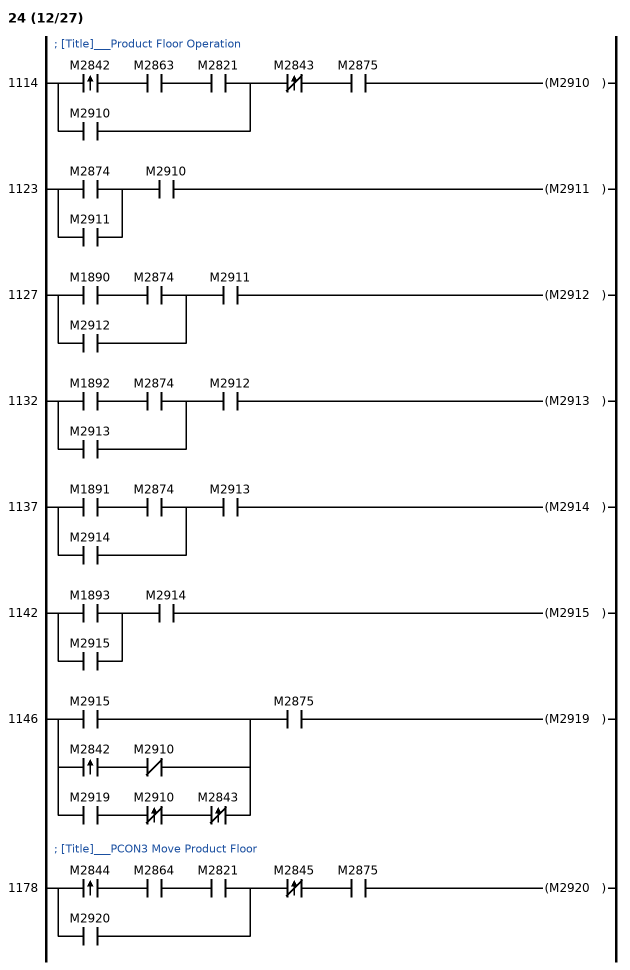
; [Title]___Product Floor Operation
1114  LDP     M2842
      AND     M2863
      AND     M2821
      OR      M2910
      ANDPI   M2843
      AND     M2875
      OUT     M2910
1123  LD      M2874
      OR      M2911
      AND     M2910
      OUT     M2911
1127  LD      M1890
      AND     M2874
      OR      M2912
      AND     M2911
      OUT     M2912
1132  LD      M1892
      AND     M2874
      OR      M2913
      AND     M2912
      OUT     M2913
1137  LD      M1891
      AND     M2874
      OR      M2914
      AND     M2913
      OUT     M2914
1142  LD      M1893
      OR      M2915
      AND     M2914
      OUT     M2915
1146  LD      M2915
      LDP     M2842
      ANI     M2910
      ORB
      LD      M2919
      ANDPI   M2910
      ANDPI   M2843
      ORB
      AND     M2875
      OUT     M2919
; [Title]___PCON3 Move Product Floor
1178  LDP     M2844
      AND     M2864
      AND     M2821
      OR      M2920
      ANDPI   M2845
      AND     M2875
      OUT     M2920
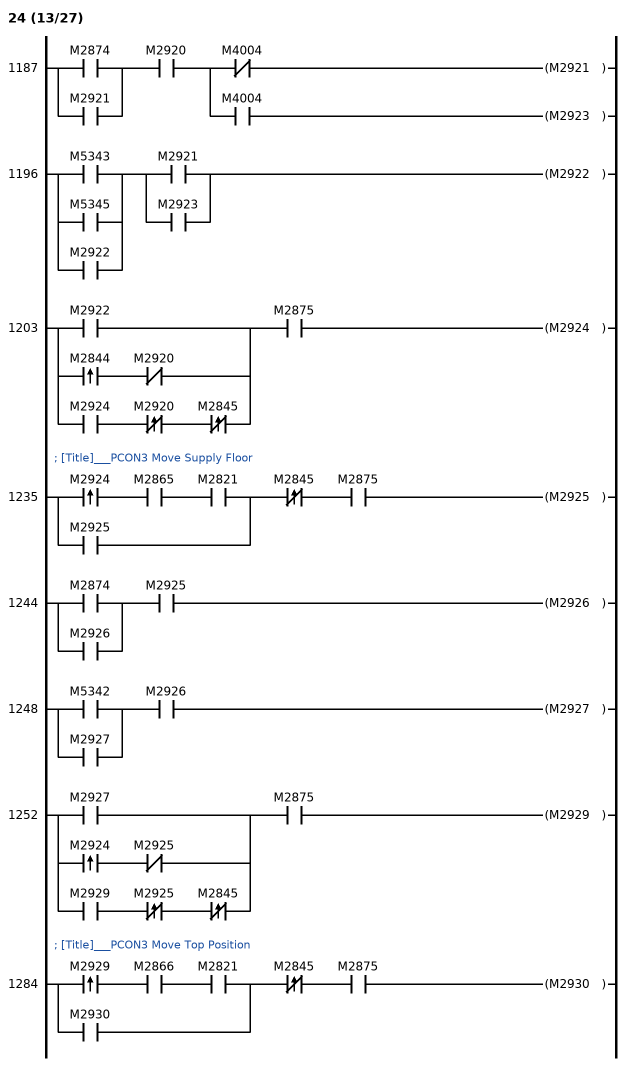
1187  LD      M2874
      OR      M2921
      AND     M2920
      MPS
      ANI     M4004
      OUT     M2921
      MPP
      AND     M4004
      OUT     M2923
1196  LD      M5343
      OR      M5345
      OR      M2922
      LD      M2921
      OR      M2923
      ANB
      OUT     M2922
1203  LD      M2922
      LDP     M2844
      ANI     M2920
      ORB
      LD      M2924
      ANDPI   M2920
      ANDPI   M2845
      ORB
      AND     M2875
      OUT     M2924
; [Title]___PCON3 Move Supply Floor
1235  LDP     M2924
      AND     M2865
      AND     M2821
      OR      M2925
      ANDPI   M2845
      AND     M2875
      OUT     M2925
1244  LD      M2874
      OR      M2926
      AND     M2925
      OUT     M2926
1248  LD      M5342
      OR      M2927
      AND     M2926
      OUT     M2927
1252  LD      M2927
      LDP     M2924
      ANI     M2925
      ORB
      LD      M2929
      ANDPI   M2925
      ANDPI   M2845
      ORB
      AND     M2875
      OUT     M2929
; [Title]___PCON3 Move Top Position
1284  LDP     M2929
      AND     M2866
      AND     M2821
      OR      M2930
      ANDPI   M2845
      AND     M2875
      OUT     M2930
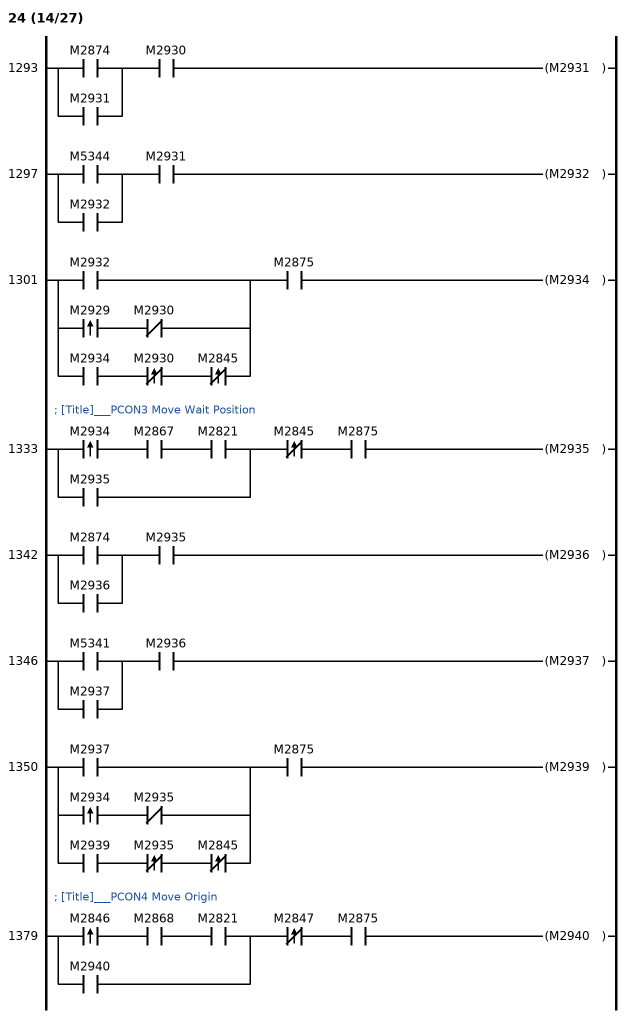
1293  LD      M2874
      OR      M2931
      AND     M2930
      OUT     M2931
1297  LD      M5344
      OR      M2932
      AND     M2931
      OUT     M2932
1301  LD      M2932
      LDP     M2929
      ANI     M2930
      ORB
      LD      M2934
      ANDPI   M2930
      ANDPI   M2845
      ORB
      AND     M2875
      OUT     M2934
; [Title]___PCON3 Move Wait Position
1333  LDP     M2934
      AND     M2867
      AND     M2821
      OR      M2935
      ANDPI   M2845
      AND     M2875
      OUT     M2935
1342  LD      M2874
      OR      M2936
      AND     M2935
      OUT     M2936
1346  LD      M5341
      OR      M2937
      AND     M2936
      OUT     M2937
1350  LD      M2937
      LDP     M2934
      ANI     M2935
      ORB
      LD      M2939
      ANDPI   M2935
      ANDPI   M2845
      ORB
      AND     M2875
      OUT     M2939
; [Title]___PCON4 Move Origin
1379  LDP     M2846
      AND     M2868
      AND     M2821
      OR      M2940
      ANDPI   M2847
      AND     M2875
      OUT     M2940
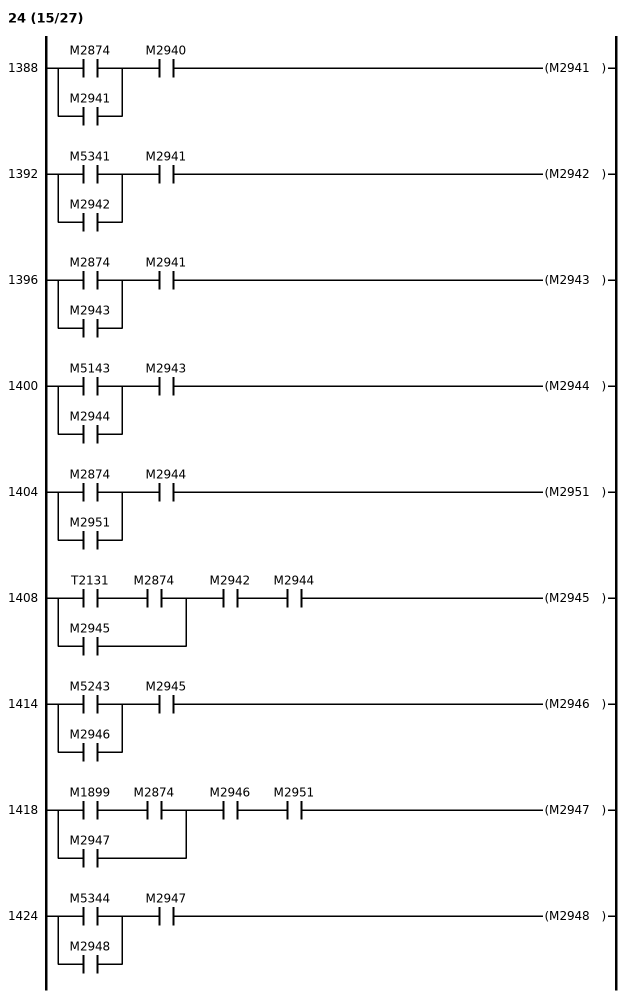
1388  LD      M2874
      OR      M2941
      AND     M2940
      OUT     M2941
1392  LD      M5341
      OR      M2942
      AND     M2941
      OUT     M2942
1396  LD      M2874
      OR      M2943
      AND     M2941
      OUT     M2943
1400  LD      M5143
      OR      M2944
      AND     M2943
      OUT     M2944
1404  LD      M2874
      OR      M2951
      AND     M2944
      OUT     M2951
1408  LD      T2131
      AND     M2874
      OR      M2945
      AND     M2942
      AND     M2944
      OUT     M2945
1414  LD      M5243
      OR      M2946
      AND     M2945
      OUT     M2946
1418  LD      M1899
      AND     M2874
      OR      M2947
      AND     M2946
      AND     M2951
      OUT     M2947
1424  LD      M5344
      OR      M2948
      AND     M2947
      OUT     M2948
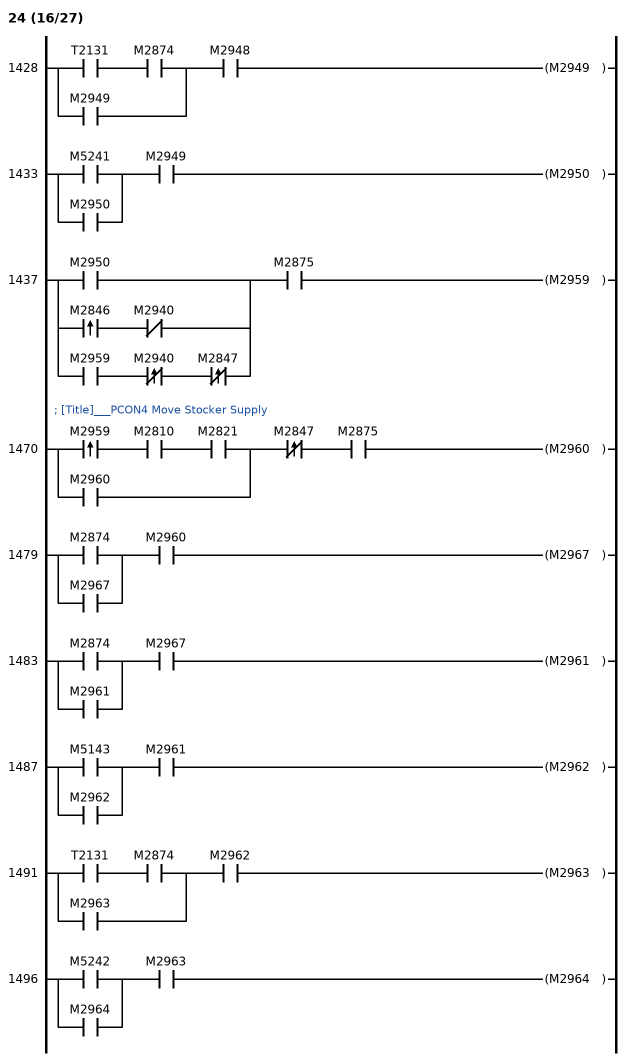
1428  LD      T2131
      AND     M2874
      OR      M2949
      AND     M2948
      OUT     M2949
1433  LD      M5241
      OR      M2950
      AND     M2949
      OUT     M2950
1437  LD      M2950
      LDP     M2846
      ANI     M2940
      ORB
      LD      M2959
      ANDPI   M2940
      ANDPI   M2847
      ORB
      AND     M2875
      OUT     M2959
; [Title]___PCON4 Move Stocker Supply
1470  LDP     M2959
      AND     M2810
      AND     M2821
      OR      M2960
      ANDPI   M2847
      AND     M2875
      OUT     M2960
1479  LD      M2874
      OR      M2967
      AND     M2960
      OUT     M2967
1483  LD      M2874
      OR      M2961
      AND     M2967
      OUT     M2961
1487  LD      M5143
      OR      M2962
      AND     M2961
      OUT     M2962
1491  LD      T2131
      AND     M2874
      OR      M2963
      AND     M2962
      OUT     M2963
1496  LD      M5242
      OR      M2964
      AND     M2963
      OUT     M2964
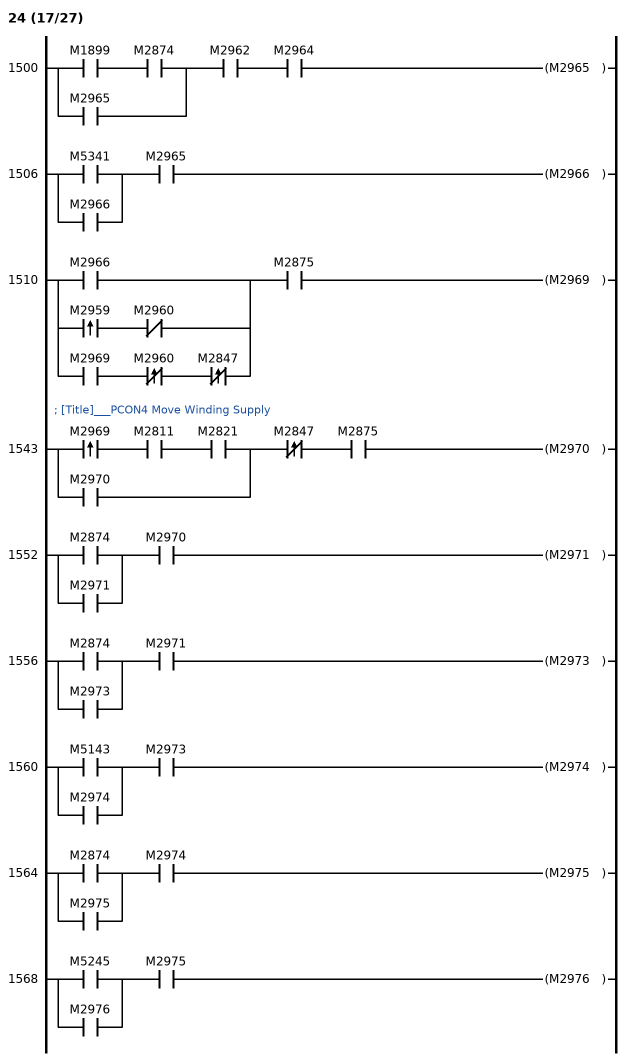
1500  LD      M1899
      AND     M2874
      OR      M2965
      AND     M2962
      AND     M2964
      OUT     M2965
1506  LD      M5341
      OR      M2966
      AND     M2965
      OUT     M2966
1510  LD      M2966
      LDP     M2959
      ANI     M2960
      ORB
      LD      M2969
      ANDPI   M2960
      ANDPI   M2847
      ORB
      AND     M2875
      OUT     M2969
; [Title]___PCON4 Move Winding Supply
1543  LDP     M2969
      AND     M2811
      AND     M2821
      OR      M2970
      ANDPI   M2847
      AND     M2875
      OUT     M2970
1552  LD      M2874
      OR      M2971
      AND     M2970
      OUT     M2971
1556  LD      M2874
      OR      M2973
      AND     M2971
      OUT     M2973
1560  LD      M5143
      OR      M2974
      AND     M2973
      OUT     M2974
1564  LD      M2874
      OR      M2975
      AND     M2974
      OUT     M2975
1568  LD      M5245
      OR      M2976
      AND     M2975
      OUT     M2976
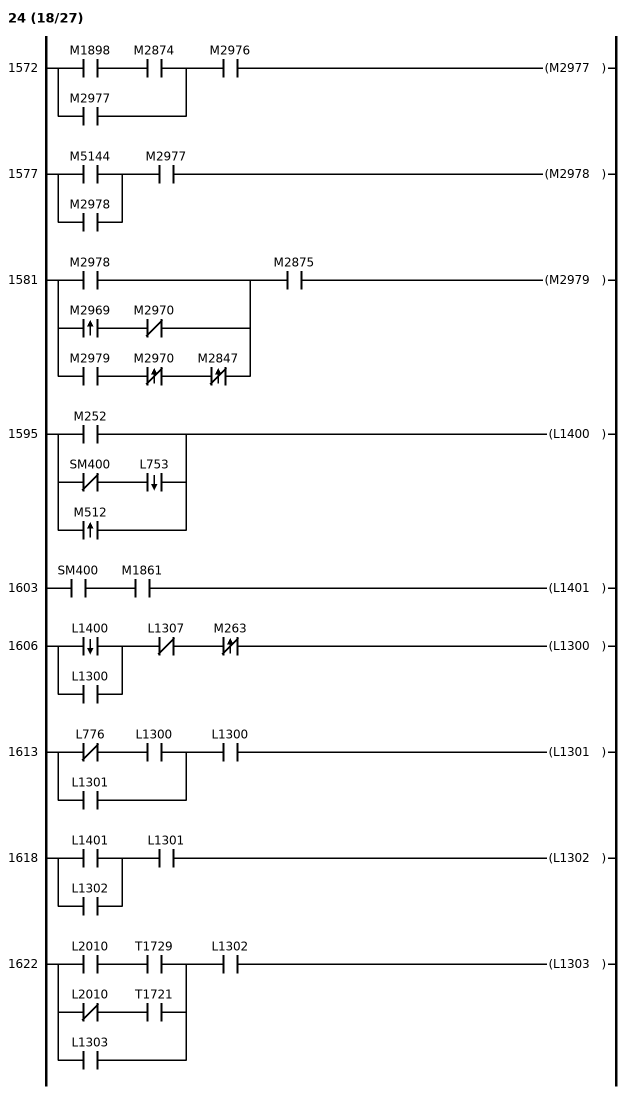
1572  LD      M1898
      AND     M2874
      OR      M2977
      AND     M2976
      OUT     M2977
1577  LD      M5144
      OR      M2978
      AND     M2977
      OUT     M2978
1581  LD      M2978
      LDP     M2969
      ANI     M2970
      ORB
      LD      M2979
      ANDPI   M2970
      ANDPI   M2847
      ORB
      AND     M2875
      OUT     M2979
; 
1595  LD      M252
      LDI     SM400
      ANDF    L753
      ORB
      ORP     M512
      OUT     L1400
1603  LD      SM400
      AND     M1861
      OUT     L1401
1606  LDF     L1400
      OR      L1300
      ANI     L1307
      ANDPI   M263
      OUT     L1300
1613  LDI     L776
      AND     L1300
      OR      L1301
      AND     L1300
      OUT     L1301
1618  LD      L1401
      OR      L1302
      AND     L1301
      OUT     L1302
1622  LD      L2010
      AND     T1729
      LDI     L2010
      AND     T1721
      ORB
      OR      L1303
      AND     L1302
      OUT     L1303
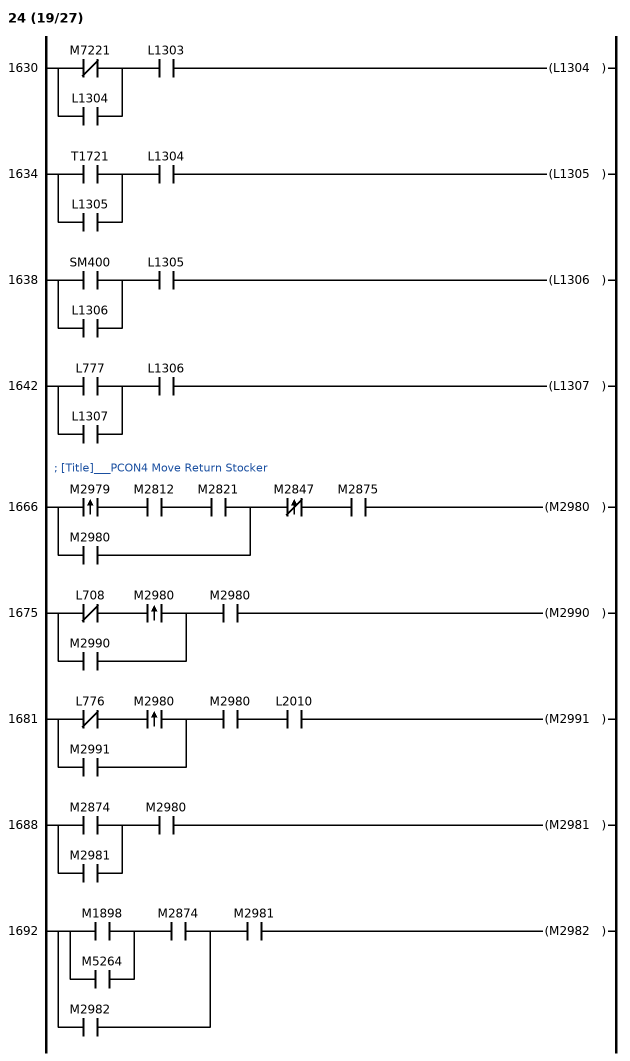
1630  LDI     M7221
      OR      L1304
      AND     L1303
      OUT     L1304
1634  LD      T1721
      OR      L1305
      AND     L1304
      OUT     L1305
1638  LD      SM400
      OR      L1306
      AND     L1305
      OUT     L1306
1642  LD      L777
      OR      L1307
      AND     L1306
      OUT     L1307
; [Title]___PCON4 Move Return Stocker
1666  LDP     M2979
      AND     M2812
      AND     M2821
      OR      M2980
      ANDPI   M2847
      AND     M2875
      OUT     M2980
1675  LDI     L708
      ANDP    M2980
      OR      M2990
      AND     M2980
      OUT     M2990
1681  LDI     L776
      ANDP    M2980
      OR      M2991
      AND     M2980
      AND     L2010
      OUT     M2991
1688  LD      M2874
      OR      M2981
      AND     M2980
      OUT     M2981
1692  LD      M1898
      OR      M5264
      AND     M2874
      OR      M2982
      AND     M2981
      OUT     M2982
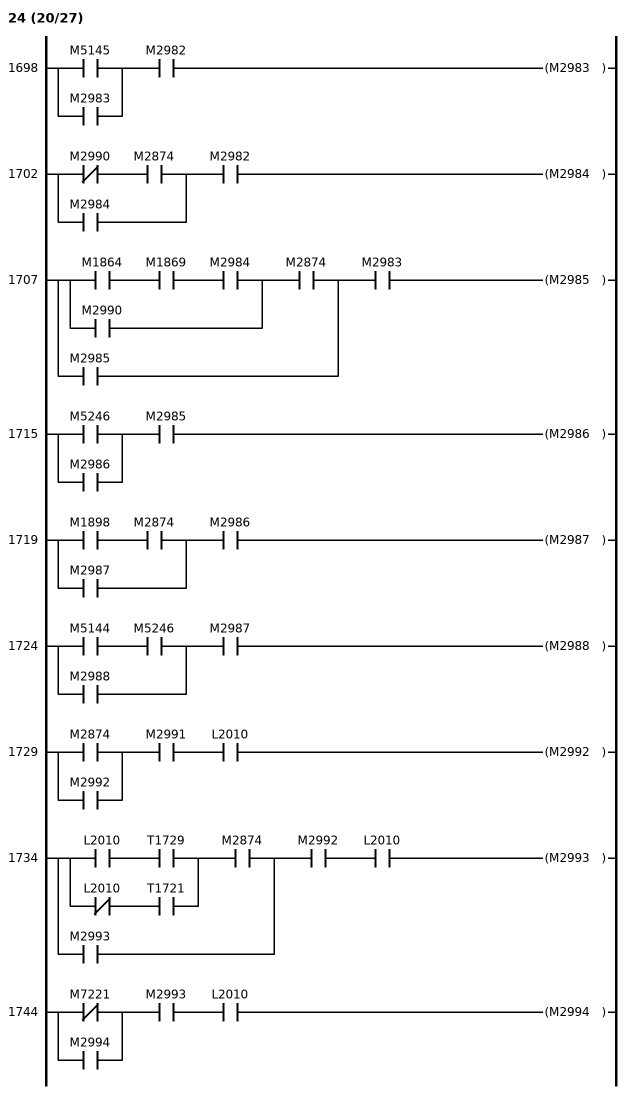
1698  LD      M5145
      OR      M2983
      AND     M2982
      OUT     M2983
1702  LDI     M2990
      AND     M2874
      OR      M2984
      AND     M2982
      OUT     M2984
1707  LD      M1864
      AND     M1869
      AND     M2984
      OR      M2990
      AND     M2874
      OR      M2985
      AND     M2983
      OUT     M2985
1715  LD      M5246
      OR      M2986
      AND     M2985
      OUT     M2986
1719  LD      M1898
      AND     M2874
      OR      M2987
      AND     M2986
      OUT     M2987
1724  LD      M5144
      AND     M5246
      OR      M2988
      AND     M2987
      OUT     M2988
1729  LD      M2874
      OR      M2992
      AND     M2991
      AND     L2010
      OUT     M2992
1734  LD      L2010
      AND     T1729
      LDI     L2010
      AND     T1721
      ORB
      AND     M2874
      OR      M2993
      AND     M2992
      AND     L2010
      OUT     M2993
1744  LDI     M7221
      OR      M2994
      AND     M2993
      AND     L2010
      OUT     M2994
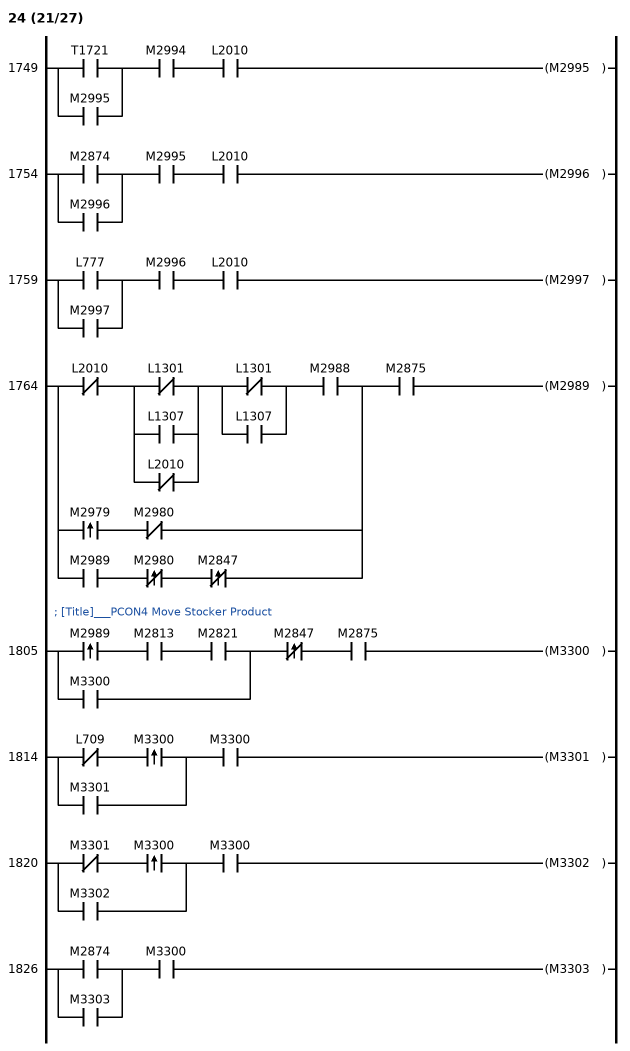
1749  LD      T1721
      OR      M2995
      AND     M2994
      AND     L2010
      OUT     M2995
1754  LD      M2874
      OR      M2996
      AND     M2995
      AND     L2010
      OUT     M2996
1759  LD      L777
      OR      M2997
      AND     M2996
      AND     L2010
      OUT     M2997
1764  LDI     L2010
      LDI     L1301
      OR      L1307
      ORI     L2010
      ANB
      LDI     L1301
      OR      L1307
      ANB
      AND     M2988
      LDP     M2979
      ANI     M2980
      ORB
      LD      M2989
      ANDPI   M2980
      ANDPI   M2847
      ORB
      AND     M2875
      OUT     M2989
; [Title]___PCON4 Move Stocker Product
1805  LDP     M2989
      AND     M2813
      AND     M2821
      OR      M3300
      ANDPI   M2847
      AND     M2875
      OUT     M3300
1814  LDI     L709
      ANDP    M3300
      OR      M3301
      AND     M3300
      OUT     M3301
1820  LDI     M3301
      ANDP    M3300
      OR      M3302
      AND     M3300
      OUT     M3302
1826  LD      M2874
      OR      M3303
      AND     M3300
      OUT     M3303
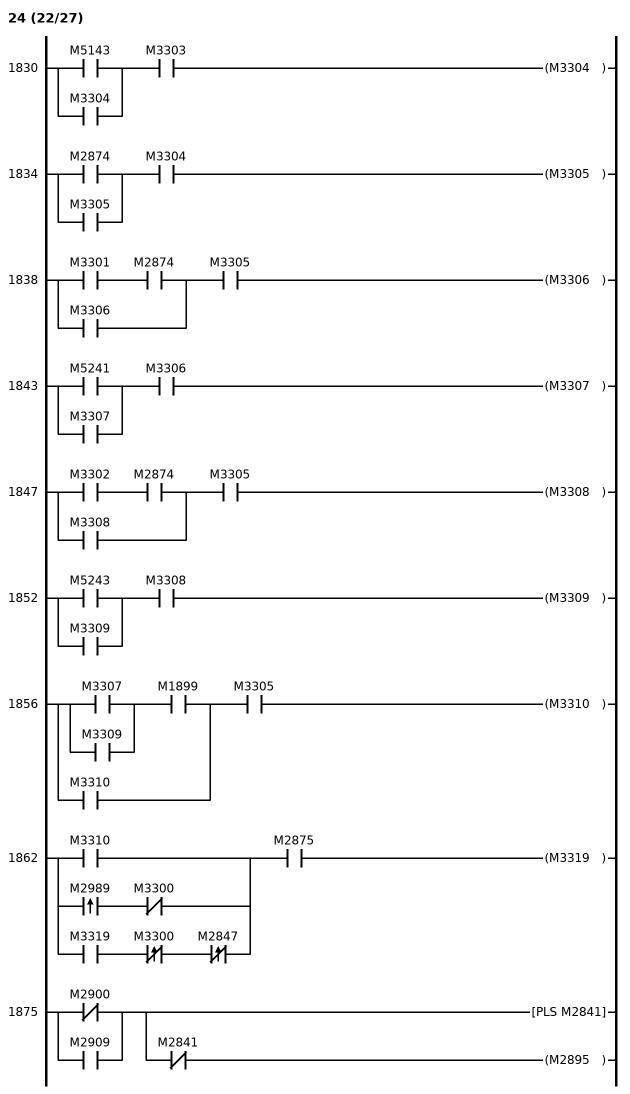
1830  LD      M5143
      OR      M3304
      AND     M3303
      OUT     M3304
1834  LD      M2874
      OR      M3305
      AND     M3304
      OUT     M3305
1838  LD      M3301
      AND     M2874
      OR      M3306
      AND     M3305
      OUT     M3306
1843  LD      M5241
      OR      M3307
      AND     M3306
      OUT     M3307
1847  LD      M3302
      AND     M2874
      OR      M3308
      AND     M3305
      OUT     M3308
1852  LD      M5243
      OR      M3309
      AND     M3308
      OUT     M3309
1856  LD      M3307
      OR      M3309
      AND     M1899
      OR      M3310
      AND     M3305
      OUT     M3310
1862  LD      M3310
      LDP     M2989
      ANI     M3300
      ORB
      LD      M3319
      ANDPI   M3300
      ANDPI   M2847
      ORB
      AND     M2875
      OUT     M3319
1875  LDI     M2900
      OR      M2909
      PLS     M2841
      ANI     M2841
      OUT     M2895
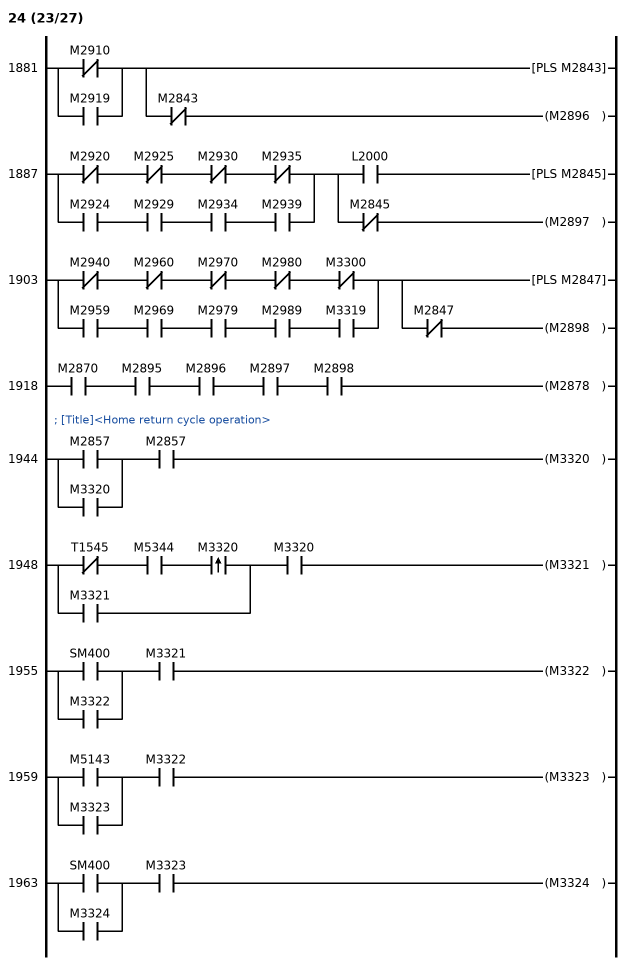
1881  LDI     M2910
      OR      M2919
      PLS     M2843
      ANI     M2843
      OUT     M2896
1887  LDI     M2920
      ANI     M2925
      ANI     M2930
      ANI     M2935
      LD      M2924
      AND     M2929
      AND     M2934
      AND     M2939
      ORB
      MPS
      AND     L2000
      PLS     M2845
      MPP
      ANI     M2845
      OUT     M2897
1903  LDI     M2940
      ANI     M2960
      ANI     M2970
      ANI     M2980
      ANI     M3300
      LD      M2959
      AND     M2969
      AND     M2979
      AND     M2989
      AND     M3319
      ORB
      PLS     M2847
      ANI     M2847
      OUT     M2898
1918  LD      M2870
      AND     M2895
      AND     M2896
      AND     M2897
      AND     M2898
      OUT     M2878
; [Title]<Home return cycle operation>
1944  LD      M2857
      OR      M3320
      AND     M2857
      OUT     M3320
1948  LDI     T1545
      AND     M5344
      ANDP    M3320
      OR      M3321
      AND     M3320
      OUT     M3321
1955  LD      SM400
      OR      M3322
      AND     M3321
      OUT     M3322
1959  LD      M5143
      OR      M3323
      AND     M3322
      OUT     M3323
1963  LD      SM400
      OR      M3324
      AND     M3323
      OUT     M3324
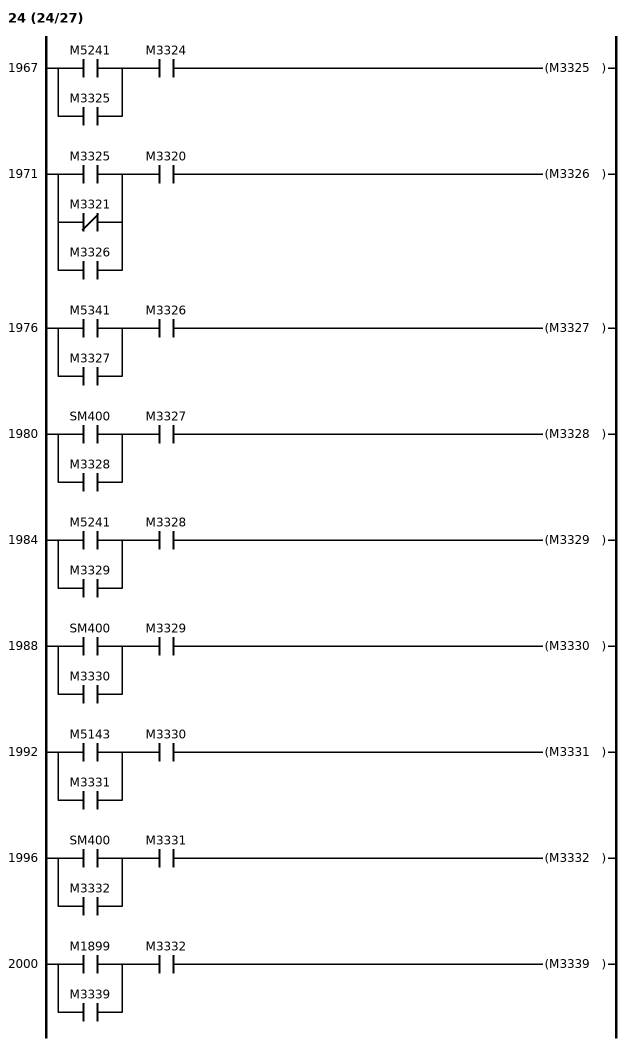
1967  LD      M5241
      OR      M3325
      AND     M3324
      OUT     M3325
1971  LD      M3325
      ORI     M3321
      OR      M3326
      AND     M3320
      OUT     M3326
1976  LD      M5341
      OR      M3327
      AND     M3326
      OUT     M3327
1980  LD      SM400
      OR      M3328
      AND     M3327
      OUT     M3328
1984  LD      M5241
      OR      M3329
      AND     M3328
      OUT     M3329
1988  LD      SM400
      OR      M3330
      AND     M3329
      OUT     M3330
1992  LD      M5143
      OR      M3331
      AND     M3330
      OUT     M3331
1996  LD      SM400
      OR      M3332
      AND     M3331
      OUT     M3332
2000  LD      M1899
      OR      M3339
      AND     M3332
      OUT     M3339
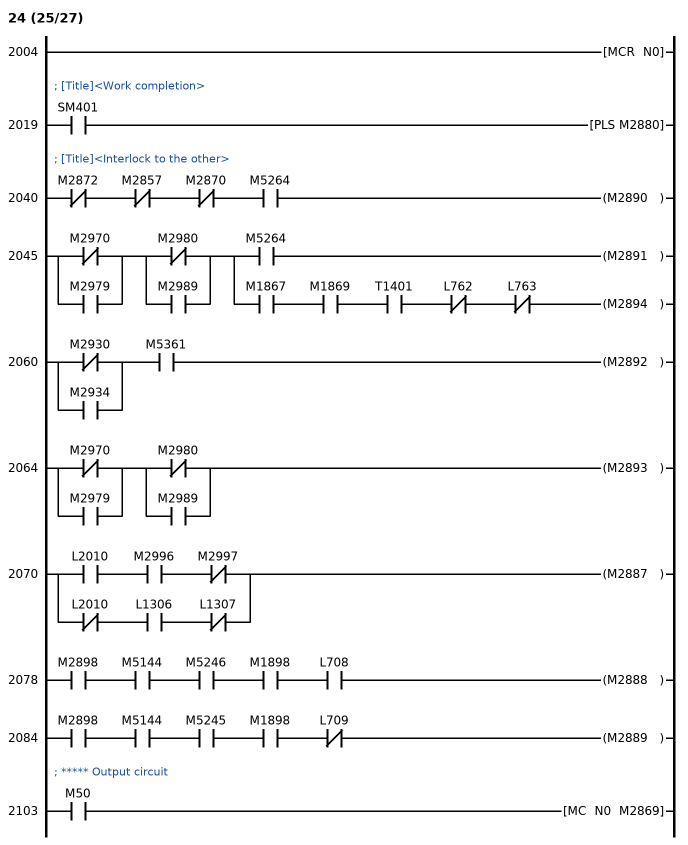
2004  MCR     N0
; [Title]<Work completion>
2019  LD      SM401
      PLS     M2880
; [Title]<Interlock to the other>
2040  LDI     M2872
      ANI     M2857
      ANI     M2870
      AND     M5264
      OUT     M2890
2045  LDI     M2970
      OR      M2979
      LDI     M2980
      OR      M2989
      ANB
      MPS
      AND     M5264
      OUT     M2891
      MPP
      AND     M1867
      AND     M1869
      AND     T1401
      ANI     L762
      ANI     L763
      OUT     M2894
2060  LDI     M2930
      OR      M2934
      AND     M5361
      OUT     M2892
2064  LDI     M2970
      OR      M2979
      LDI     M2980
      OR      M2989
      ANB
      OUT     M2893
2070  LD      L2010
      AND     M2996
      ANI     M2997
      LDI     L2010
      AND     L1306
      ANI     L1307
      ORB
      OUT     M2887
2078  LD      M2898
      AND     M5144
      AND     M5246
      AND     M1898
      AND     L708
      OUT     M2888
2084  LD      M2898
      AND     M5144
      AND     M5245
      AND     M1898
      ANI     L709
      OUT     M2889
; ***** Output circuit
2103  LD      M50
      MC      N0 M2869
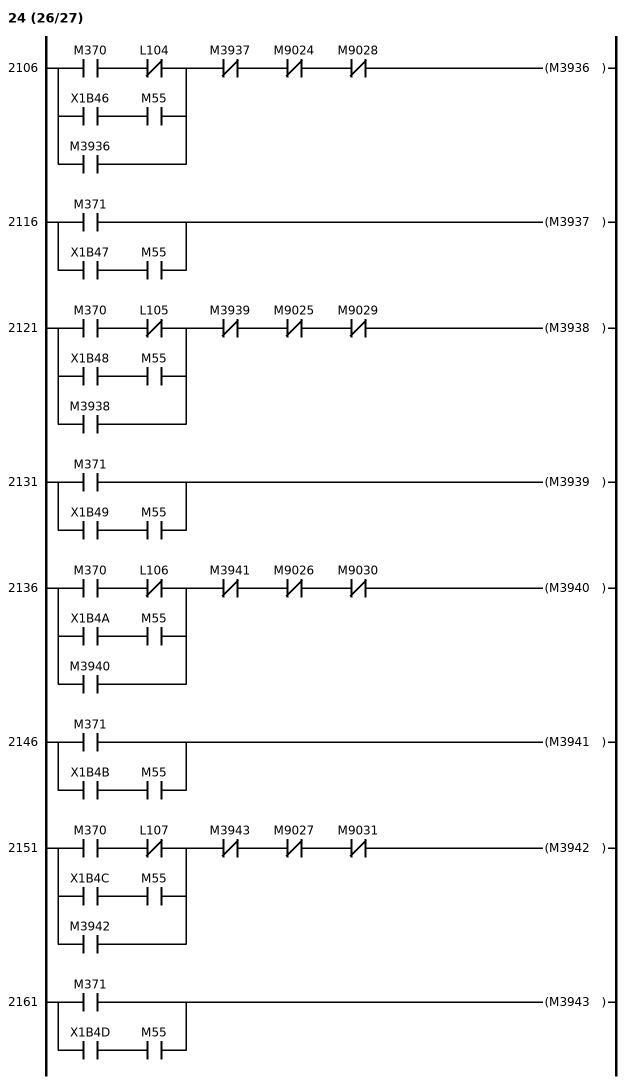
2106  LD      M370
      ANI     L104
      LD      X1B46
      AND     M55
      ORB
      OR      M3936
      ANI     M3937
      ANI     M9024
      ANI     M9028
      OUT     M3936
2116  LD      M371
      LD      X1B47
      AND     M55
      ORB
      OUT     M3937
2121  LD      M370
      ANI     L105
      LD      X1B48
      AND     M55
      ORB
      OR      M3938
      ANI     M3939
      ANI     M9025
      ANI     M9029
      OUT     M3938
2131  LD      M371
      LD      X1B49
      AND     M55
      ORB
      OUT     M3939
2136  LD      M370
      ANI     L106
      LD      X1B4A
      AND     M55
      ORB
      OR      M3940
      ANI     M3941
      ANI     M9026
      ANI     M9030
      OUT     M3940
2146  LD      M371
      LD      X1B4B
      AND     M55
      ORB
      OUT     M3941
2151  LD      M370
      ANI     L107
      LD      X1B4C
      AND     M55
      ORB
      OR      M3942
      ANI     M3943
      ANI     M9027
      ANI     M9031
      OUT     M3942
2161  LD      M371
      LD      X1B4D
      AND     M55
      ORB
      OUT     M3943
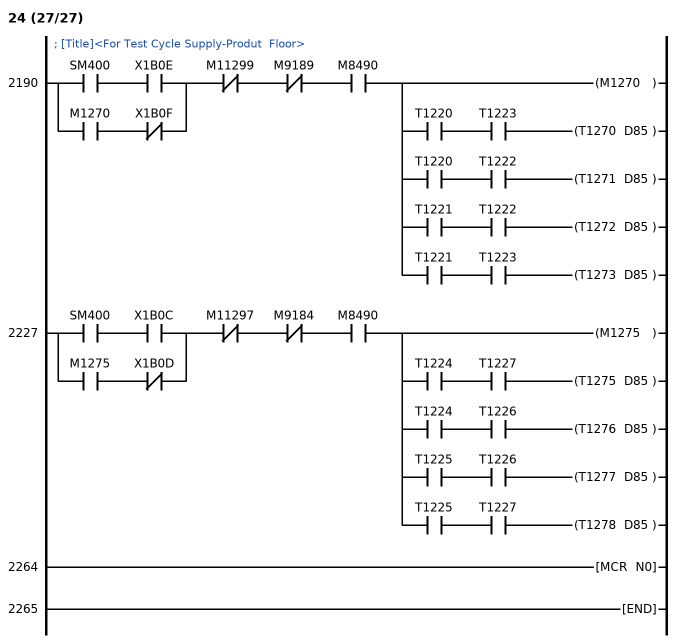
; [Title]<For Test Cycle Supply-Produt  Floor>
2190  LD      SM400
      AND     X1B0E
      LD      M1270
      ANI     X1B0F
      ORB
      ANI     M11299
      ANI     M9189
      AND     M8490
      OUT     M1270
      MPS
      AND     T1220
      AND     T1223
      OUT     T1270 D85
      MRD
      AND     T1220
      AND     T1222
      OUT     T1271 D85
      MRD
      AND     T1221
      AND     T1222
      OUT     T1272 D85
      MPP
      AND     T1221
      AND     T1223
      OUT     T1273 D85
2227  LD      SM400
      AND     X1B0C
      LD      M1275
      ANI     X1B0D
      ORB
      ANI     M11297
      ANI     M9184
      AND     M8490
      OUT     M1275
      MPS
      AND     T1224
      AND     T1227
      OUT     T1275 D85
      MRD
      AND     T1224
      AND     T1226
      OUT     T1276 D85
      MRD
      AND     T1225
      AND     T1226
      OUT     T1277 D85
      MPP
      AND     T1225
      AND     T1227
      OUT     T1278 D85
2264  MCR     N0
2265  END
END_PROGRAM

PROGRAM 25
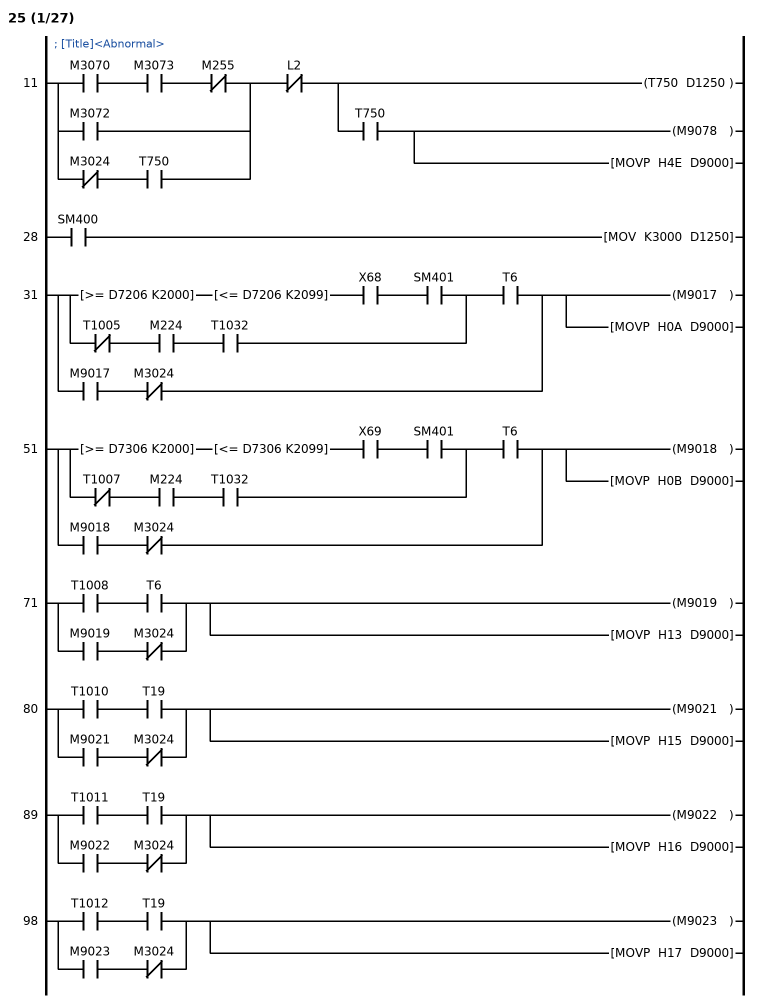
; [Title]<Abnormal>
11    LD      M3070
      AND     M3073
      ANI     M255
      OR      M3072
      LDI     M3024
      AND     T750
      ORB
      ANI     L2
      OUT     T750 D1250
      AND     T750
      OUT     M9078
      MOVP    H4E D9000
28    LD      SM400
      MOV     K3000 D1250
31    LD>=    D7206 K2000
      AND<=   D7206 K2099
      AND     X68
      AND     SM401
      LDI     T1005
      AND     M224
      AND     T1032
      ORB
      AND     T6
      LD      M9017
      ANI     M3024
      ORB
      OUT     M9017
      MOVP    H0A D9000
51    LD>=    D7306 K2000
      AND<=   D7306 K2099
      AND     X69
      AND     SM401
      LDI     T1007
      AND     M224
      AND     T1032
      ORB
      AND     T6
      LD      M9018
      ANI     M3024
      ORB
      OUT     M9018
      MOVP    H0B D9000
71    LD      T1008
      AND     T6
      LD      M9019
      ANI     M3024
      ORB
      OUT     M9019
      MOVP    H13 D9000
80    LD      T1010
      AND     T19
      LD      M9021
      ANI     M3024
      ORB
      OUT     M9021
      MOVP    H15 D9000
89    LD      T1011
      AND     T19
      LD      M9022
      ANI     M3024
      ORB
      OUT     M9022
      MOVP    H16 D9000
98    LD      T1012
      AND     T19
      LD      M9023
      ANI     M3024
      ORB
      OUT     M9023
      MOVP    H17 D9000
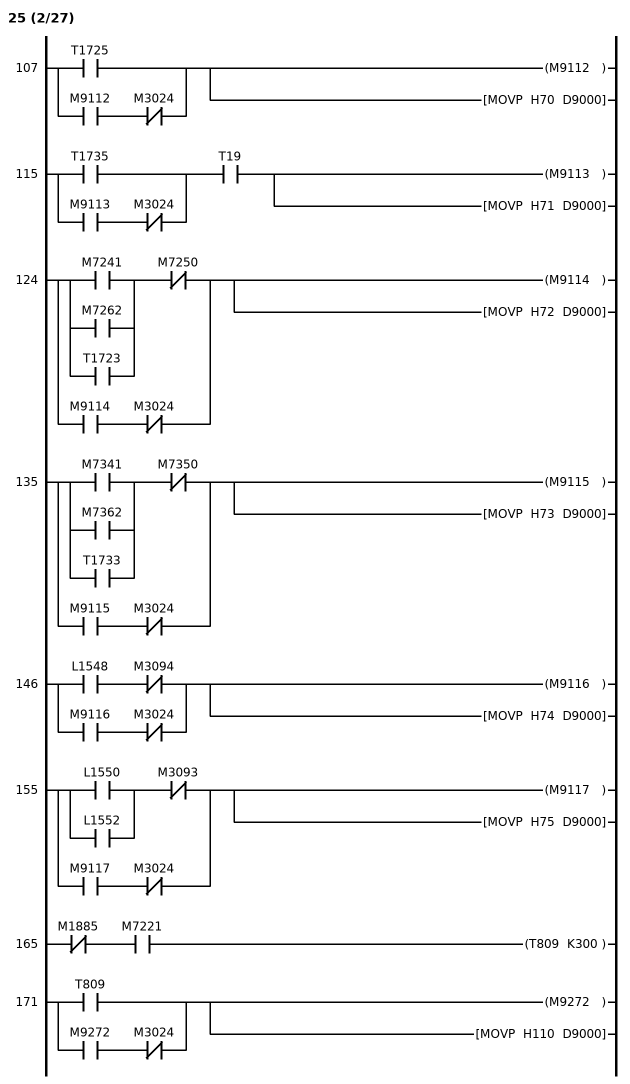
107   LD      T1725
      LD      M9112
      ANI     M3024
      ORB
      OUT     M9112
      MOVP    H70 D9000
115   LD      T1735
      LD      M9113
      ANI     M3024
      ORB
      AND     T19
      OUT     M9113
      MOVP    H71 D9000
124   LD      M7241
      OR      M7262
      OR      T1723
      ANI     M7250
      LD      M9114
      ANI     M3024
      ORB
      OUT     M9114
      MOVP    H72 D9000
135   LD      M7341
      OR      M7362
      OR      T1733
      ANI     M7350
      LD      M9115
      ANI     M3024
      ORB
      OUT     M9115
      MOVP    H73 D9000
146   LD      L1548
      ANI     M3094
      LD      M9116
      ANI     M3024
      ORB
      OUT     M9116
      MOVP    H74 D9000
155   LD      L1550
      OR      L1552
      ANI     M3093
      LD      M9117
      ANI     M3024
      ORB
      OUT     M9117
      MOVP    H75 D9000
165   LDI     M1885
      AND     M7221
      OUT     T809 K300
171   LD      T809
      LD      M9272
      ANI     M3024
      ORB
      OUT     M9272
      MOVP    H110 D9000
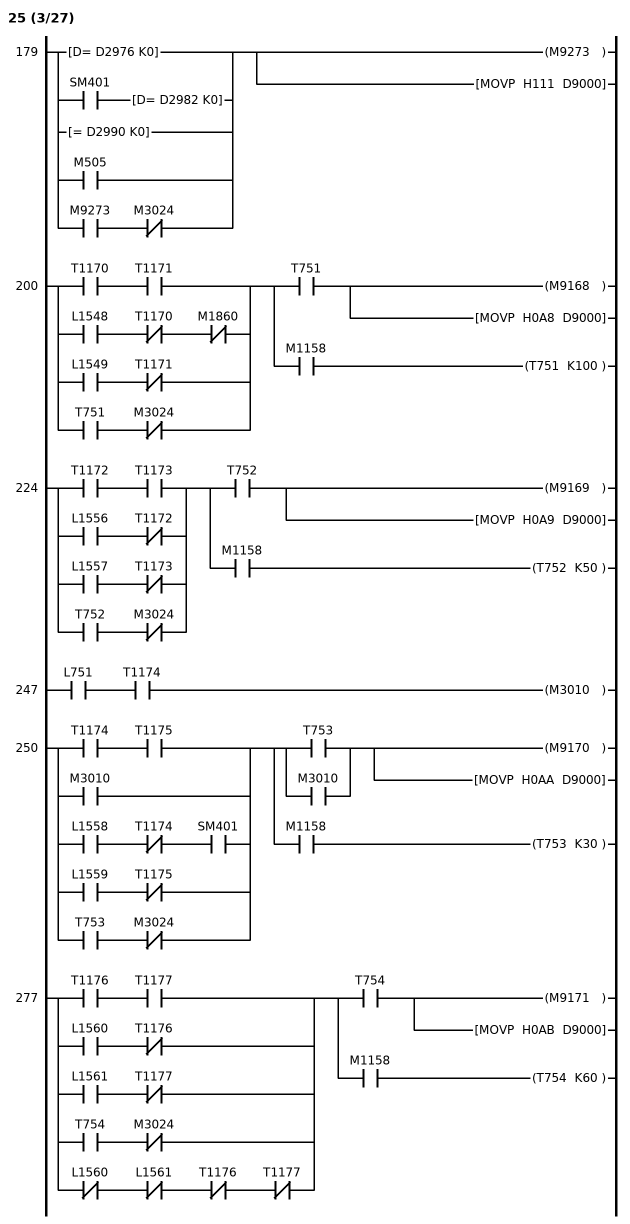
179   LDD=    D2976 K0
      LD      SM401
      ANDD=   D2982 K0
      ORB
      OR=     D2990 K0
      OR      M505
      LD      M9273
      ANI     M3024
      ORB
      OUT     M9273
      MOVP    H111 D9000
200   LD      T1170
      AND     T1171
      LD      L1548
      ANI     T1170
      ANI     M1860
      ORB
      LD      L1549
      ANI     T1171
      ORB
      LD      T751
      ANI     M3024
      ORB
      MPS
      AND     T751
      OUT     M9168
      MOVP    H0A8 D9000
      MPP
      AND     M1158
      OUT     T751 K100
224   LD      T1172
      AND     T1173
      LD      L1556
      ANI     T1172
      ORB
      LD      L1557
      ANI     T1173
      ORB
      LD      T752
      ANI     M3024
      ORB
      MPS
      AND     T752
      OUT     M9169
      MOVP    H0A9 D9000
      MPP
      AND     M1158
      OUT     T752 K50
247   LD      L751
      AND     T1174
      OUT     M3010
250   LD      T1174
      AND     T1175
      OR      M3010
      LD      L1558
      ANI     T1174
      AND     SM401
      ORB
      LD      L1559
      ANI     T1175
      ORB
      LD      T753
      ANI     M3024
      ORB
      MPS
      LD      T753
      OR      M3010
      ANB
      OUT     M9170
      MOVP    H0AA D9000
      MPP
      AND     M1158
      OUT     T753 K30
277   LD      T1176
      AND     T1177
      LD      L1560
      ANI     T1176
      ORB
      LD      L1561
      ANI     T1177
      ORB
      LD      T754
      ANI     M3024
      ORB
      LDI     L1560
      ANI     L1561
      ANI     T1176
      ANI     T1177
      ORB
      MPS
      AND     T754
      OUT     M9171
      MOVP    H0AB D9000
      MPP
      AND     M1158
      OUT     T754 K60
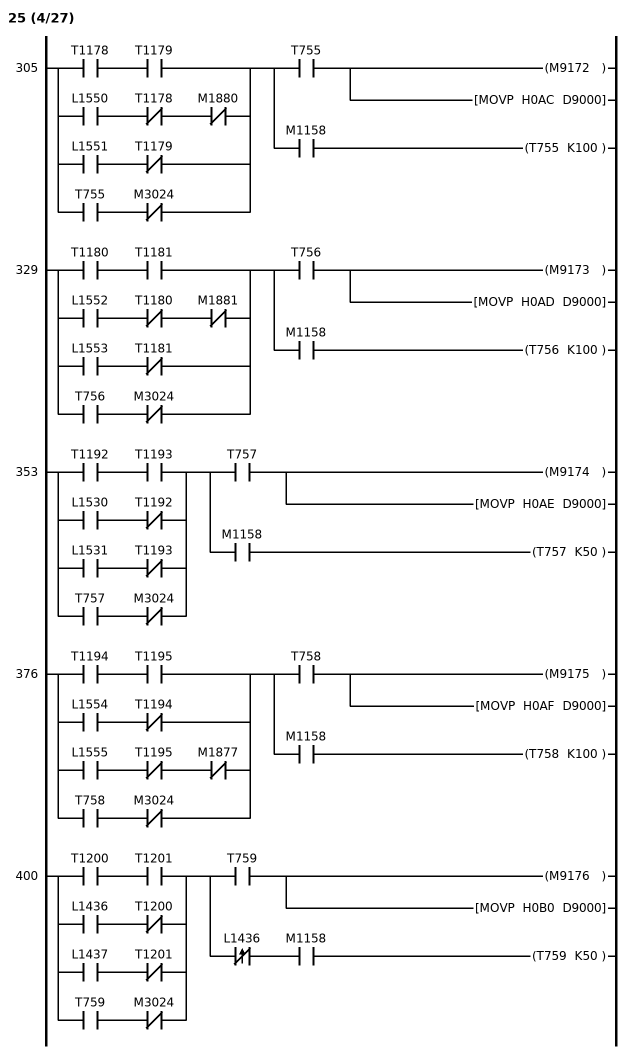
305   LD      T1178
      AND     T1179
      LD      L1550
      ANI     T1178
      ANI     M1880
      ORB
      LD      L1551
      ANI     T1179
      ORB
      LD      T755
      ANI     M3024
      ORB
      MPS
      AND     T755
      OUT     M9172
      MOVP    H0AC D9000
      MPP
      AND     M1158
      OUT     T755 K100
329   LD      T1180
      AND     T1181
      LD      L1552
      ANI     T1180
      ANI     M1881
      ORB
      LD      L1553
      ANI     T1181
      ORB
      LD      T756
      ANI     M3024
      ORB
      MPS
      AND     T756
      OUT     M9173
      MOVP    H0AD D9000
      MPP
      AND     M1158
      OUT     T756 K100
353   LD      T1192
      AND     T1193
      LD      L1530
      ANI     T1192
      ORB
      LD      L1531
      ANI     T1193
      ORB
      LD      T757
      ANI     M3024
      ORB
      MPS
      AND     T757
      OUT     M9174
      MOVP    H0AE D9000
      MPP
      AND     M1158
      OUT     T757 K50
376   LD      T1194
      AND     T1195
      LD      L1554
      ANI     T1194
      ORB
      LD      L1555
      ANI     T1195
      ANI     M1877
      ORB
      LD      T758
      ANI     M3024
      ORB
      MPS
      AND     T758
      OUT     M9175
      MOVP    H0AF D9000
      MPP
      AND     M1158
      OUT     T758 K100
400   LD      T1200
      AND     T1201
      LD      L1436
      ANI     T1200
      ORB
      LD      L1437
      ANI     T1201
      ORB
      LD      T759
      ANI     M3024
      ORB
      MPS
      AND     T759
      OUT     M9176
      MOVP    H0B0 D9000
      MPP
      ANDPI   L1436
      AND     M1158
      OUT     T759 K50
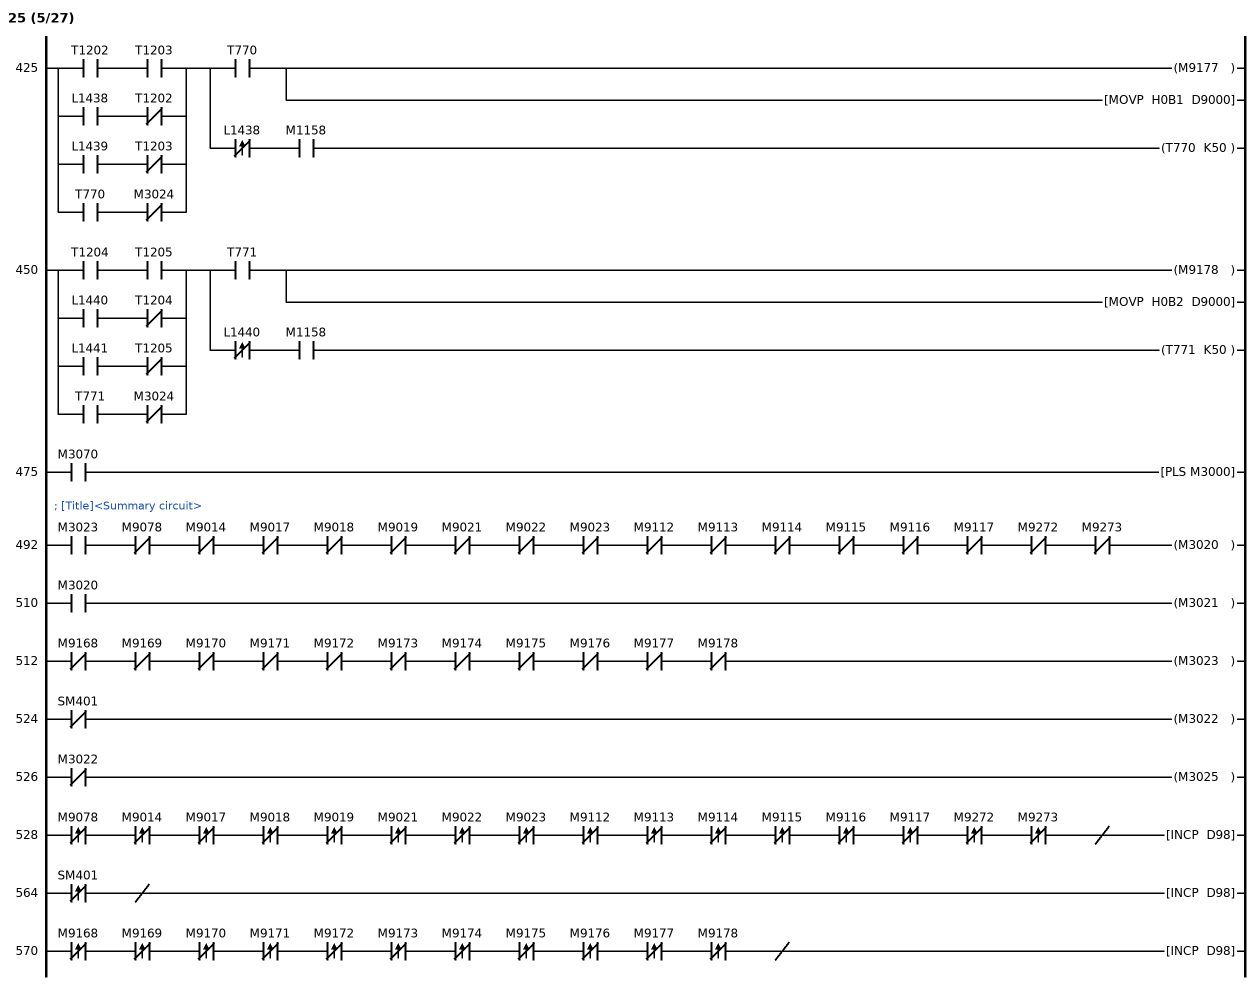
425   LD      T1202
      AND     T1203
      LD      L1438
      ANI     T1202
      ORB
      LD      L1439
      ANI     T1203
      ORB
      LD      T770
      ANI     M3024
      ORB
      MPS
      AND     T770
      OUT     M9177
      MOVP    H0B1 D9000
      MPP
      ANDPI   L1438
      AND     M1158
      OUT     T770 K50
450   LD      T1204
      AND     T1205
      LD      L1440
      ANI     T1204
      ORB
      LD      L1441
      ANI     T1205
      ORB
      LD      T771
      ANI     M3024
      ORB
      MPS
      AND     T771
      OUT     M9178
      MOVP    H0B2 D9000
      MPP
      ANDPI   L1440
      AND     M1158
      OUT     T771 K50
475   LD      M3070
      PLS     M3000
; [Title]<Summary circuit>
492   LD      M3023
      ANI     M9078
      ANI     M9014
      ANI     M9017
      ANI     M9018
      ANI     M9019
      ANI     M9021
      ANI     M9022
      ANI     M9023
      ANI     M9112
      ANI     M9113
      ANI     M9114
      ANI     M9115
      ANI     M9116
      ANI     M9117
      ANI     M9272
      ANI     M9273
      OUT     M3020
510   LD      M3020
      OUT     M3021
512   LDI     M9168
      ANI     M9169
      ANI     M9170
      ANI     M9171
      ANI     M9172
      ANI     M9173
      ANI     M9174
      ANI     M9175
      ANI     M9176
      ANI     M9177
      ANI     M9178
      OUT     M3023
524   LDI     SM401
      OUT     M3022
526   LDI     M3022
      OUT     M3025
528   LDPI    M9078
      ANDPI   M9014
      ANDPI   M9017
      ANDPI   M9018
      ANDPI   M9019
      ANDPI   M9021
      ANDPI   M9022
      ANDPI   M9023
      ANDPI   M9112
      ANDPI   M9113
      ANDPI   M9114
      ANDPI   M9115
      ANDPI   M9116
      ANDPI   M9117
      ANDPI   M9272
      ANDPI   M9273
      INV
      INCP    D98
564   LDPI    SM401
      INV
      INCP    D98
570   LDPI    M9168
      ANDPI   M9169
      ANDPI   M9170
      ANDPI   M9171
      ANDPI   M9172
      ANDPI   M9173
      ANDPI   M9174
      ANDPI   M9175
      ANDPI   M9176
      ANDPI   M9177
      ANDPI   M9178
      INV
      INCP    D98
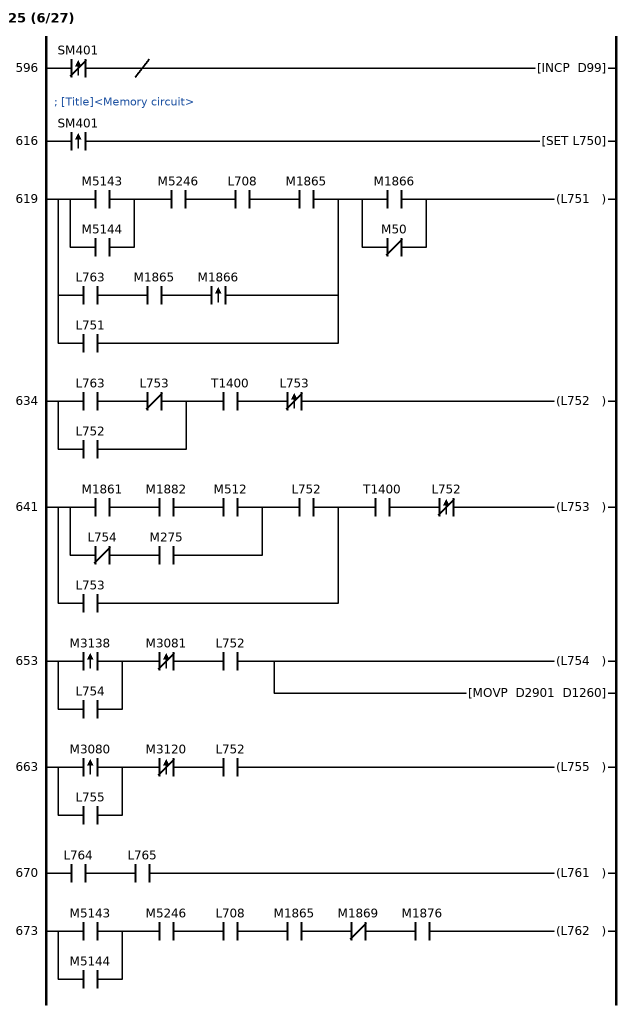
596   LDPI    SM401
      INV
      INCP    D99
; [Title]<Memory circuit>
616   LDP     SM401
      SET     L750
619   LD      M5143
      OR      M5144
      AND     M5246
      AND     L708
      AND     M1865
      LD      L763
      AND     M1865
      ANDP    M1866
      ORB
      OR      L751
      LD      M1866
      ORI     M50
      ANB
      OUT     L751
634   LD      L763
      ANI     L753
      OR      L752
      AND     T1400
      ANDPI   L753
      OUT     L752
641   LD      M1861
      AND     M1882
      AND     M512
      LDI     L754
      AND     M275
      ORB
      AND     L752
      OR      L753
      AND     T1400
      ANDPI   L752
      OUT     L753
653   LDP     M3138
      OR      L754
      ANDPI   M3081
      AND     L752
      OUT     L754
      MOVP    D2901 D1260
663   LDP     M3080
      OR      L755
      ANDPI   M3120
      AND     L752
      OUT     L755
670   LD      L764
      AND     L765
      OUT     L761
673   LD      M5143
      OR      M5144
      AND     M5246
      AND     L708
      AND     M1865
      ANI     M1869
      AND     M1876
      OUT     L762
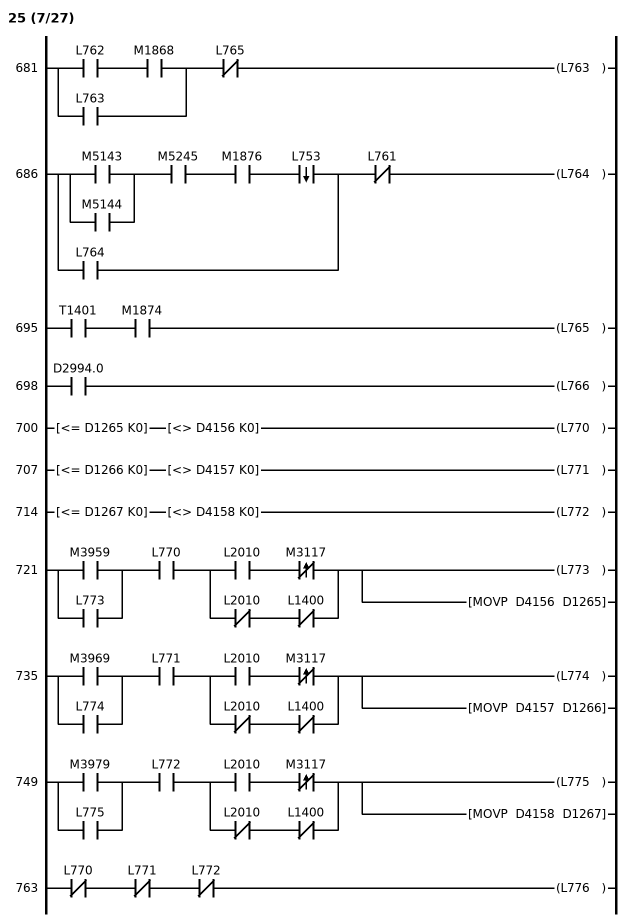
681   LD      L762
      AND     M1868
      OR      L763
      ANI     L765
      OUT     L763
686   LD      M5143
      OR      M5144
      AND     M5245
      AND     M1876
      ANDF    L753
      OR      L764
      ANI     L761
      OUT     L764
695   LD      T1401
      AND     M1874
      OUT     L765
698   LD      D2994.0
      OUT     L766
700   LD<=    D1265 K0
      AND<>   D4156 K0
      OUT     L770
707   LD<=    D1266 K0
      AND<>   D4157 K0
      OUT     L771
714   LD<=    D1267 K0
      AND<>   D4158 K0
      OUT     L772
721   LD      M3959
      OR      L773
      AND     L770
      LD      L2010
      ANDPI   M3117
      LDI     L2010
      ANI     L1400
      ORB
      ANB
      OUT     L773
      MOVP    D4156 D1265
735   LD      M3969
      OR      L774
      AND     L771
      LD      L2010
      ANDPI   M3117
      LDI     L2010
      ANI     L1400
      ORB
      ANB
      OUT     L774
      MOVP    D4157 D1266
749   LD      M3979
      OR      L775
      AND     L772
      LD      L2010
      ANDPI   M3117
      LDI     L2010
      ANI     L1400
      ORB
      ANB
      OUT     L775
      MOVP    D4158 D1267
763   LDI     L770
      ANI     L771
      ANI     L772
      OUT     L776
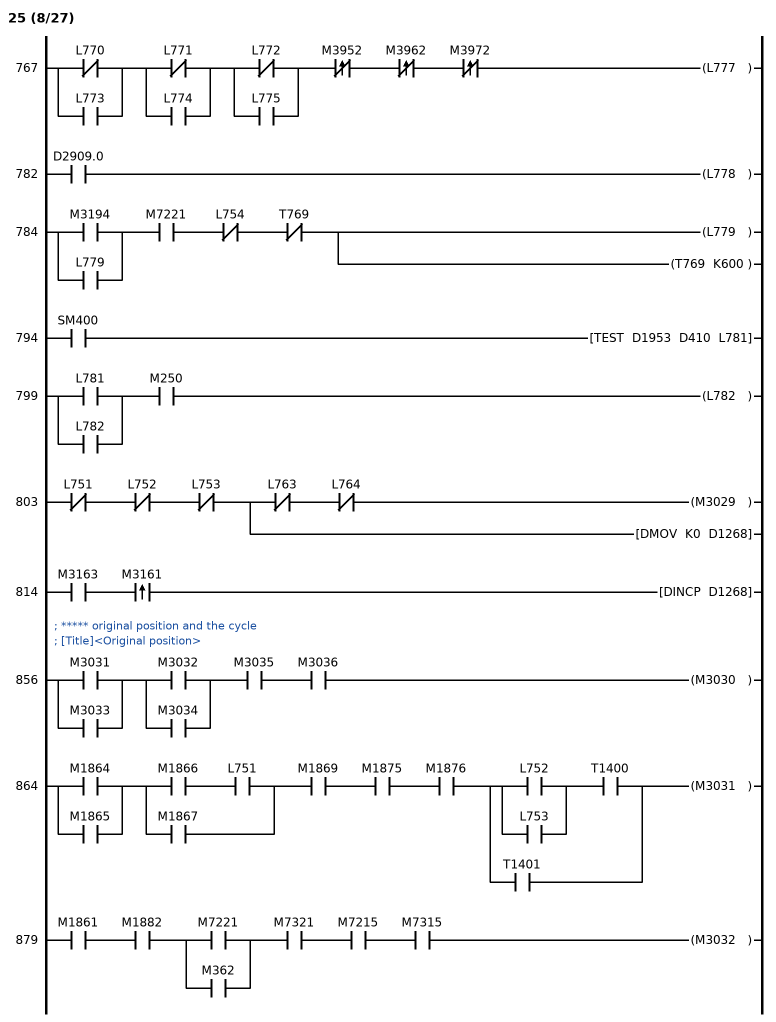
767   LDI     L770
      OR      L773
      LDI     L771
      OR      L774
      ANB
      LDI     L772
      OR      L775
      ANB
      ANDPI   M3952
      ANDPI   M3962
      ANDPI   M3972
      OUT     L777
782   LD      D2909.0
      OUT     L778
784   LD      M3194
      OR      L779
      AND     M7221
      ANI     L754
      ANI     T769
      OUT     L779
      OUT     T769 K600
794   LD      SM400
      TEST    D1953 D410 L781
799   LD      L781
      OR      L782
      AND     M250
      OUT     L782
803   LDI     L751
      ANI     L752
      ANI     L753
      MPS
      ANI     L763
      ANI     L764
      OUT     M3029
      MPP
      DMOV    K0 D1268
814   LD      M3163
      ANDP    M3161
      DINCP   D1268
; ***** original position and the cycle
; [Title]<Original position>
856   LD      M3031
      OR      M3033
      LD      M3032
      OR      M3034
      ANB
      AND     M3035
      AND     M3036
      OUT     M3030
864   LD      M1864
      OR      M1865
      LD      M1866
      AND     L751
      OR      M1867
      ANB
      AND     M1869
      AND     M1875
      AND     M1876
      LD      L752
      OR      L753
      AND     T1400
      OR      T1401
      ANB
      OUT     M3031
879   LD      M1861
      AND     M1882
      LD      M7221
      OR      M362
      ANB
      AND     M7321
      AND     M7215
      AND     M7315
      OUT     M3032
